{attribute 'GeneratedUsingTerminal: EL2564-0000-0016'}
{attribute addProperty BoxType "EL2564-0000-0016"}
{attribute addProperty Id "PWM_Inputs_Channel_1AT %I*PWM_Inputs_Channel_304DC2453PWM_Inputs_Channel_2AT %I*PWM_Inputs_Channel_304DC2453PWM_Inputs_Channel_3AT %I*PWM_Inputs_Channel_304DC2453PWM_Inputs_Channel_4AT %I*PWM_Inputs_Channel_304DC2453PWM_Outputs_Channel_1AT %Q*PWM_Outputs_Channel_D6F04FBD2PWM_Outputs_Channel_2AT %Q*PWM_Outputs_Channel_D6F04FBD2PWM_Outputs_Channel_3AT %Q*PWM_Outputs_Channel_D6F04FBD2PWM_Outputs_Channel_4AT %Q*PWM_Outputs_Channel_D6F04FBD2WcStateAT %I*WcState_9091E0EB2InfoDataAT %I*InfoData_32EB74EA10"}
{attribute addProperty CRC "407469422"}
{attribute addProperty Size "32"}
TYPE EL2564_18497D6E EXTENDS EtcSlaveTerminalBase_947E5A46 :
STRUCT
	{attribute addProperty Name "PWM_Inputs_Channel_1"}
	PWM_Inputs_Channel_1 : PWM_Inputs_Channel_304DC245;
	{attribute addProperty Name "PWM_Inputs_Channel_2"}
	PWM_Inputs_Channel_2 : PWM_Inputs_Channel_304DC245;
	{attribute addProperty Name "PWM_Inputs_Channel_3"}
	PWM_Inputs_Channel_3 : PWM_Inputs_Channel_304DC245;
	{attribute addProperty Name "PWM_Inputs_Channel_4"}
	PWM_Inputs_Channel_4 : PWM_Inputs_Channel_304DC245;
	{attribute addProperty Name "PWM_Outputs_Channel_1"}
	PWM_Outputs_Channel_1 : PWM_Outputs_Channel_D6F04FBD;
	{attribute addProperty Name "PWM_Outputs_Channel_2"}
	PWM_Outputs_Channel_2 : PWM_Outputs_Channel_D6F04FBD;
	{attribute addProperty Name "PWM_Outputs_Channel_3"}
	PWM_Outputs_Channel_3 : PWM_Outputs_Channel_D6F04FBD;
	{attribute addProperty Name "PWM_Outputs_Channel_4"}
	PWM_Outputs_Channel_4 : PWM_Outputs_Channel_D6F04FBD;
	{attribute addProperty Name "WcState"}
	WcState : WcState_9091E0EB;
	{attribute addProperty Name "InfoData"}
	InfoData : InfoData_32EB74EA;
END_STRUCT
END_TYPE

(* stored: Version 1.2.0.0, ProductVersion 3.1.4024.9
   DUT EL2564_18497D6E: Id {3af6dfdc-a6a1-495a-9411-82c11e0a96cb} *)
